DATA_BLOCK "ChangeOver_DB"
VAR
  Robot_1 : STRUCT
    Req_RobotToMaintenancePos : Bool;
    Req_RobotToHomePos : Bool;
    Sensor_3 : Bool;
    Sensor_4 : Bool;
    Sensor_5 : Bool;
    Sensor_6 : Bool;
    Sensor_7 : Bool;
    Sensor_8 : Bool;
    EmptyProcess : Bool;
    EmptyFinish : Bool;
    Spare : Bool;
    HMI_MaintenancePosReqSel : Bool;
    HMI_MaintenancePosActive : Bool;
    MaintenancePosReqSelFlag : Bool;
    HMI_MaintenanceHomeReq : Bool;
    NoTaskRunning : Bool;
    Spare_6 : Bool;
    Step : Int;
  END_STRUCT;
  Robot_2 : STRUCT
    Req_RobotToMaintenancePos : Bool;
    Req_RobotToHomePos : Bool;
    Sensor_3 : Bool;
    Sensor_4 : Bool;
    Sensor_5 : Bool;
    Sensor_6 : Bool;
    Sensor_7 : Bool;
    Sensor_8 : Bool;
    EmptyProcess : Bool;
    EmptyFinish : Bool;
    Spare : Bool;
    HMI_MaintenancePosReqSel : Bool;
    HMI_MaintenancePosActive : Bool;
    MaintenancePosReqSelFlag : Bool;
    HMI_MaintenanceHomeReq : Bool;
    NoTaskRunning : Bool;
    Spare_6 : Bool;
    Step : Int;
  END_STRUCT;
  Robot_3 : STRUCT
    Req_RobotToMaintenancePos : Bool;
    Req_RobotToHomePos : Bool;
    Sensor_3 : Bool;
    Sensor_4 : Bool;
    Sensor_5 : Bool;
    Sensor_6 : Bool;
    Sensor_7 : Bool;
    Sensor_8 : Bool;
    EmptyProcess : Bool;
    EmptyFinish : Bool;
    Spare : Bool;
    HMI_MaintenancePosReqSel : Bool;
    HMI_MaintenancePosActive : Bool;
    MaintenancePosReqSelFlag : Bool;
    HMI_MaintenanceHomeReq : Bool;
    NoTaskRunning : Bool;
    Spare_6 : Bool;
    Step : Int;
  END_STRUCT;
  H_Line : STRUCT
    Sensor_1 : Bool;
    Sensor_2 : Bool;
    Sensor_3 : Bool;
    Sensor_4 : Bool;
    Sensor_5 : Bool;
    Sensor_6 : Bool;
    Sensor_7 : Bool;
    Sensor_8 : Bool;
    Sensor_9 : Bool;
    Sensor_10 : Bool;
    Sensor_11 : Bool;
    Sensor_12 : Bool;
    Sensor_13 : Bool;
    Sensor_14 : Bool;
    Sensor_15 : Bool;
    Sensor_16 : Bool;
    EmptyProcess : Bool;
    EmptyFinish : Bool;
    Spare : Bool;
    Spare_1 : Bool;
    Spare_2 : Bool;
    Spare_3 : Bool;
    Spare_4 : Bool;
    Spare_5 : Bool;
    Spare_6 : Bool;
    Step : Int;
  END_STRUCT;
  J_Line : STRUCT
    Sensor_1 : Bool;
    Sensor_2 : Bool;
    Sensor_3 : Bool;
    Sensor_4 : Bool;
    Sensor_5 : Bool;
    Sensor_6 : Bool;
    Sensor_7 : Bool;
    Sensor_8 : Bool;
    Sensor_9 : Bool;
    Sensor_10 : Bool;
    Sensor_11 : Bool;
    Sensor_12 : Bool;
    Sensor_13 : Bool;
    Sensor_14 : Bool;
    Sensor_15 : Bool;
    Sensor_16 : Bool;
    EmptyProcess : Bool;
    EmptyFinish : Bool;
    Spare : Bool;
    Spare_1 : Bool;
    Spare_2 : Bool;
    Spare_3 : Bool;
    Spare_4 : Bool;
    Spare_5 : Bool;
    Spare_6 : Bool;
    Step : Int;
  END_STRUCT;
  K_Line : STRUCT
    Sensor_1 : Bool;
    Sensor_2 : Bool;
    Sensor_3 : Bool;
    Sensor_4 : Bool;
    Sensor_5 : Bool;
    Sensor_6 : Bool;
    Sensor_7 : Bool;
    Sensor_8 : Bool;
    Sensor_9 : Bool;
    Sensor_10 : Bool;
    Sensor_11 : Bool;
    Sensor_12 : Bool;
    Sensor_13 : Bool;
    Sensor_14 : Bool;
    Sensor_15 : Bool;
    Sensor_16 : Bool;
    EmptyProcess : Bool;
    EmptyFinish : Bool;
    Spare : Bool;
    Spare_1 : Bool;
    Spare_2 : Bool;
    Spare_3 : Bool;
    Spare_4 : Bool;
    Spare_5 : Bool;
    Spare_6 : Bool;
    Step : Int;
  END_STRUCT;
  L_Line : STRUCT
    Sensor_1 : Bool;
    Sensor_2 : Bool;
    Sensor_3 : Bool;
    Sensor_4 : Bool;
    Sensor_5 : Bool;
    Sensor_6 : Bool;
    Sensor_7 : Bool;
    Sensor_8 : Bool;
    Sensor_9 : Bool;
    Sensor_10 : Bool;
    Sensor_11 : Bool;
    Sensor_12 : Bool;
    Sensor_13 : Bool;
    Sensor_14 : Bool;
    Sensor_15 : Bool;
    Sensor_16 : Bool;
    EmptyProcess : Bool;
    EmptyFinish : Bool;
    Spare : Bool;
    Spare_1 : Bool;
    Spare_2 : Bool;
    Spare_3 : Bool;
    Spare_4 : Bool;
    Spare_5 : Bool;
    Spare_6 : Bool;
    Step : Int;
  END_STRUCT;
  Global : STRUCT
    AllFixtureScanCompareOk : Bool;
    ChangeOverRequest : Bool;
    ChangeOverToolScanFlag : Bool;
    ManualModeFlag : Bool;
    ScanFixtureFlag : Bool;
    Station_empty : Bool;
    ChangeOverSelected : Bool;
    ScanFixtureFlag_ChangeOver : Bool;
    A1_TableScanStart : Bool;
    A2_TableScanStart : Bool;
    Hmi_Confirm_ChangeOver : Bool;
    ChangeOverActive : Bool;
    Hmi_ForceChangeOver : Bool;
    Spare_13 : Bool;
    Spare_14 : Bool;
    Spare_15 : Bool;
  END_STRUCT;
  P : Array[0..20] of Bool;
  Time : Array[0..3] of TOF_TIME;
  Robot1 : STRUCT
    Ring1Weight : Int;
    ShaftWeight : Int;
    MagnetWeight : Int;
    Ring2Weight : Int;
  END_STRUCT;
  Robot2 : STRUCT
    Ring1Weight : Int;
    ShaftWeight : Int;
    MagnetWeight : Int;
    Ring2Weight : Int;
  END_STRUCT;
  Robot3 : STRUCT
    Ring1Weight : Int;
    ShaftWeight : Int;
    MagnetWeight : Int;
    Ring2Weight : Int;
  END_STRUCT;
END_VAR
BEGIN
END_DATA_BLOCK
